# B&R Automation Studio project Genmot_Markalama_ (part 5)

#### GRYAxisControl.c - Implementation code
```c
/*******************************************************************
 * COPYRIGHT -- Bernecker + Rainer
 ********************************************************************
 * PROGRAM: Basic
 * File: Basic.c
 * Author: Bernecker + Rainer
 * Created: December 01, 2009
 ********************************************************************
 * Implementation of Program Basic
 ********************************************************************/

#ifdef _DEFAULT_INCLUDES
#include <AsDefault.h>
#endif
#include <string.h>

/* defines of the state-constants */
#define STATE_WAIT              0
#define STATE_POWER_ON          1
#define STATE_HOME              2

#define STATE_READY             10
#define STATE_HALT              11
#define STATE_STOP              12
#define STATE_JOG_POSITIVE      13
#define STATE_JOG_NEGATIVE      14
#define STATE_MOVE_ABSOLUTE     15
#define STATE_MOVE_ADDITIVE     16
#define STATE_MOVE_VELOCITY     17

#define STATE_ERROR_AXIS        100
#define STATE_ERROR             101
#define STATE_ERROR_RESET       102
#define STATE_READ              103

_LOCAL REAL   data;

_INIT void GRYAxis_init(void)
{

	/* get axis object */
	Axis1Obj = (UDINT)&GRY_Axis;

	AxisStep = STATE_WAIT;  /* start step */

	GRYAxis.Parameter.Velocity              = 10000;  /*velocity for movement*/
	GRYAxis.Parameter.Acceleration          = 40000;  /*acceleration for movement*/
	GRYAxis.Parameter.Deceleration          = 40000;  /*deceleration for movement*/
	GRYAxis.Parameter.JogVelocity           = 10000;   /*velocity for jogging */

}

_CYCLIC void GRYAxis_cyclic(void)
{
	if(GRYAxis.Command.Power)
	{
		GRYAxis.Speed.VelocityOverride			= 1.0;
	}

/***************************************************************
        Control Sequence
***************************************************************/

/* status information is read before the step sequencer to attain a shorter reaction time */
/************************ MC_READSTATUS *************************/
	MC_ReadStatus_0.Enable = !MC_ReadStatus_0.Error;
	MC_ReadStatus_0.Axis = Axis1Obj;
	MC_ReadStatus(&MC_ReadStatus_0);
	GRYAxis.AxisState.Disabled             = MC_ReadStatus_0.Disabled;
	GRYAxis.AxisState.StandStill           = MC_ReadStatus_0.StandStill;
	GRYAxis.AxisState.Stopping             = MC_ReadStatus_0.Stopping;
	GRYAxis.AxisState.Homing               = MC_ReadStatus_0.Homing;
	GRYAxis.AxisState.DiscreteMotion       = MC_ReadStatus_0.DiscreteMotion;
	GRYAxis.AxisState.ContinuousMotion     = MC_ReadStatus_0.ContinuousMotion;
	GRYAxis.AxisState.SynchronizedMotion   = MC_ReadStatus_0.SynchronizedMotion;
	GRYAxis.AxisState.ErrorStop            = MC_ReadStatus_0.Errorstop;

	/********************MC_BR_READDRIVESTATUS***********************/
	MC_BR_ReadDriveStatus_0.Enable = !MC_BR_ReadDriveStatus_0.Error;
	MC_BR_ReadDriveStatus_0.Axis = Axis1Obj;
	MC_BR_ReadDriveStatus_0.AdrDriveStatus = (UDINT)&(GRYAxis.Status.DriveStatus);
	MC_BR_ReadDriveStatus(&MC_BR_ReadDriveStatus_0);

	/******************** MC_READACTUALPOSITION *********************/
	MC_ReadActualPosition_0.Enable = (!MC_ReadActualPosition_0.Error);
	MC_ReadActualPosition_0.Axis = Axis1Obj;
	MC_ReadActualPosition(&MC_ReadActualPosition_0);
	if(MC_ReadActualPosition_0.Valid == 1)
	{
		GRYAxis.Status.ActPosition = MC_ReadActualPosition_0.Position;
	}

	/******************** MC_READACTUALVELOCITY *********************/
	MC_ReadActualVelocity_0.Enable = (!MC_ReadActualVelocity_0.Error);
	MC_ReadActualVelocity_0.Axis = Axis1Obj;
	MC_ReadActualVelocity(&MC_ReadActualVelocity_0);
	if(MC_ReadActualVelocity_0.Valid == 1)
	{
		GRYAxis.Status.ActVelocity = MC_ReadActualVelocity_0.Velocity;
	}

	/*********************** MC SET OVERRIDE *********************/
	MC_SetOverride_0.Enable = (!MC_SetOverride_0.Error);
	MC_SetOverride_0.AccFactor = GRYAxis.Speed.AccelerationOverride = 1.0;
	if ((GRYAxis.Speed.VelocityOverride < 2.01) && (GRYAxis.Speed.VelocityOverride > 0.0000001))
	{
		MC_SetOverride_0.VelFactor = GRYAxis.Speed.VelocityOverride;
	}
	MC_SetOverride_0.Axis=Axis1Obj;
	MC_SetOverride(&MC_SetOverride_0);

	/************************ MC_READAXISERROR **********************/
	MC_ReadAxisError_0.Enable = !MC_ReadAxisError_0.Error;
	MC_ReadAxisError_0.Axis = Axis1Obj;
	MC_ReadAxisError_0.DataAddress = (UDINT)&(GRYAxis.Status.ErrorText);
	MC_ReadAxisError_0.DataLength = sizeof(GRYAxis.Status.ErrorText);
	strcpy((void*)&MC_ReadAxisError_0.DataObjectName,"acp10etxen");
	MC_ReadAxisError(&MC_ReadAxisError_0);

	/* central monitoring of stop command attains a shorter reaction time in case of emergency stop */
	/******************CHECK for STOP COMMAND************************/
	if (GRYAxis.Command.Stop == 1)
	{
		if ((AxisStep >= STATE_READY) && (AxisStep < STATE_ERROR))
		{
			/* reset all FB execute inputs we use */
			MC_Home_0.Execute = 0;
			MC_Stop_0.Execute = 0;
			MC_MoveAbsolute_0.Execute = 0;
			MC_MoveAdditive_0.Execute = 0;
			MC_MoveVelocity_0.Execute = 0;
			MC_ReadAxisError_0.Acknowledge = 0;
			MC_Reset_0.Execute = 0;

			/* reset user commands */
			GRYAxis.Command.Stop = 0;
			GRYAxis.Command.Home = 0;
			GRYAxis.Command.MoveJogPos = 0;
			GRYAxis.Command.MoveJogNeg = 0;
			GRYAxis.Command.MoveVelocity = 0;
			GRYAxis.Command.MoveAbsolute = 0;
			GRYAxis.Command.MoveAdditive = 0;
			AxisStep = STATE_STOP;
		}
	}

	/**************** CHECK FOR GENERAL AXIS ERROR ******************/
	if ((MC_ReadAxisError_0.AxisErrorID != 0) && (MC_ReadAxisError_0.Valid == 1))
	{
		AxisStep = STATE_ERROR_AXIS;
	}
		/***************** CHECK IF POWER SHOULD BE OFF *******************/
	else if ((GRYAxis.Command.Power == 0) && (MC_ReadAxisError_0.Valid == 1))
	{
		if ((MC_ReadStatus_0.Errorstop == 1) && (MC_ReadStatus_0.Valid == 1))
		{
			AxisStep = STATE_ERROR_RESET;
		}
		else
		{
			AxisStep = STATE_WAIT;
		}
	}

	switch(AxisStep)
	{
		/******************** WAIT *************************/
		case STATE_WAIT:  /* STATE: Wait */
			if (GRYAxis.Command.Power == 1)
			{
				AxisStep = STATE_POWER_ON;
			}
			else
			{
				MC_Power_0.Enable = 0;

			}

			/* reset all FB execute inputs we use */
			MC_Home_0.Execute = 0;
			MC_Stop_0.Execute = 0;
			MC_MoveAbsolute_0.Execute = 0;
			MC_MoveAdditive_0.Execute = 0;
			MC_MoveVelocity_0.Execute = 0;
			MC_ReadAxisError_0.Acknowledge = 0;
			MC_Reset_0.Execute = 0;

			/* reset user commands */
			GRYAxis.Command.Stop = 0;
			GRYAxis.Command.Home = 0;
			GRYAxis.Command.MoveJogPos = 0;
			GRYAxis.Command.MoveJogNeg = 0;
			GRYAxis.Command.MoveVelocity = 0;
			GRYAxis.Command.MoveAbsolute = 0;
			GRYAxis.Command.MoveAdditive = 0;

			GRYAxis.Status.ErrorID = 0;
			break;

		/******************** POWER ON **********************/
		case STATE_POWER_ON:  /* STATE: Power on */
			MC_Power_0.Enable = 1;
			if (MC_Power_0.Status == 1)
			{
			if (!GRXHomeOk)
			{
			GRYAxis.Command.Home = 1;
			}
			AxisStep = STATE_READY;
			}
			/* if a power error occured go to error state */
			if (MC_Power_0.Error == 1)
			{
				GRYAxis.Status.ErrorID = MC_Power_0.ErrorID;
				AxisStep = STATE_ERROR;
			}
			break;

		/******************** READY **********************/
		case STATE_READY:  /* STATE: Waiting for commands */
			if (GRYAxis.Command.Home == 1)
			{
				GRYAxis.Command.Home = 0;
				AxisStep = STATE_HOME;
			}
			else if (GRYAxis.Command.Stop == 1)
			{
				AxisStep = STATE_STOP;
			}
			else if (GRYAxis.Command.MoveJogPos == 1)
			{
				AxisStep = STATE_JOG_POSITIVE;
			}
			else if (GRYAxis.Command.MoveJogNeg == 1)
			{
				AxisStep = STATE_JOG_NEGATIVE;
			}
			else if (GRYAxis.Command.MoveAbsolute == 1)
			{
				GRYAxis.Command.MoveAbsolute = 0;
				AxisStep = STATE_MOVE_ABSOLUTE;
			}
			else if (GRYAxis.Command.MoveAdditive == 1)
			{
				GRYAxis.Command.MoveAdditive = 0;
				AxisStep = STATE_MOVE_ADDITIVE;
			}
			else if (GRYAxis.Command.MoveVelocity == 1)
			{
				GRYAxis.Command.MoveVelocity = 0;
				AxisStep = STATE_MOVE_VELOCITY;
			}
			else if (GRYAxis.Command.Halt == 1)
			{
				GRYAxis.Command.Halt = 0;
				AxisStep = STATE_HALT;
			}
			break;

		/******************** HOME **********************/
		case STATE_HOME:  /* STATE: start homing process */
			MC_Home_0.Position = GRYAxis.Parameter.HomePosition;
			MC_Home_0.HomingMode = GRYAxis.Parameter.HomeMode;
			MC_Home_0.Execute = 1;
			if (MC_Home_0.Done == 1)
			{

				MC_Home_0.Execute = 0;
				AxisStep = STATE_READ;
			}
			/* if a homing error occured go to error state */
			if (MC_Home_0.Error == 1)
			{
				MC_Home_0.Execute = 0;
				GRYAxis.Status.ErrorID = MC_Home_0.ErrorID;
				AxisStep = STATE_ERROR;
			}
			break;

		/************************HALT MOVEMENT**************************/
		case STATE_HALT:  /* STATE: Stop the active movement */
			MC_Halt_0.Deceleration = GRYAxis.Parameter.Deceleration;
			MC_Halt_0.Execute = 1;
			if (MC_Halt_0.Done == 1)
			{
				MC_Halt_0.Execute = 0;
				AxisStep = STATE_READY;
			}
			/*check if error occured */
			if (MC_Halt_0.Error == 1)
			{
				MC_Halt_0.Execute = 0;
				GRYAxis.Status.ErrorID = MC_Halt_0.ErrorID;
				AxisStep = STATE_ERROR;
			}
			break;

		/*********************** STOP MOVEMENT *************************/
		case STATE_STOP: /* STATE: Stop movement as long as command is set */
			MC_Stop_0.Deceleration = GRYAxis.Parameter.Deceleration;
			MC_Stop_0.Execute = 1;
			/* if axis is stopped go to ready state */
			if ((MC_Stop_0.Done == 1) && (GRYAxis.Command.Stop == 0))
			{
				MC_Stop_0.Execute = 0;
				AxisStep = STATE_READY;
			}
			/* check if error occured */
			if (MC_Stop_0.Error == 1)
			{
				GRYAxis.Status.ErrorID = MC_Stop_0.ErrorID;
				MC_Stop_0.Execute = 0;
				AxisStep = STATE_ERROR;
			}
			break;

		/******************** START JOG MOVEMENT POSITVE **********************/
		case STATE_JOG_POSITIVE:  /* STATE: Start jog movement in positive direction */
			MC_MoveVelocity_0.Velocity      = GRYAxis.Parameter.JogVelocity;
			MC_MoveVelocity_0.Acceleration  = GRYAxis.Parameter.Acceleration;
			MC_MoveVelocity_0.Deceleration  = GRYAxis.Parameter.Deceleration;
			MC_MoveVelocity_0.Direction     = mcPOSITIVE_DIR;
			MC_MoveVelocity_0.Execute = 1;
			/* check if jog movement should be stopped */
			if (GRYAxis.Command.MoveJogPos == 0)
			{
				MC_MoveVelocity_0.Execute = 0;
				AxisStep = STATE_HALT;
			}
			/* check if error occured */
			if (MC_MoveVelocity_0.Error == 1)
			{
				GRYAxis.Status.ErrorID = MC_MoveVelocity_0.ErrorID;
				MC_MoveVelocity_0.Execute = 0;
				AxisStep = STATE_ERROR;
			}
			break;

		/******************** START JOG MOVEMENT NEGATIVE **********************/
		case STATE_JOG_NEGATIVE:  /* STATE: Start jog movement in negative direction */
			MC_MoveVelocity_0.Velocity      = GRYAxis.Parameter.JogVelocity;
			MC_MoveVelocity_0.Acceleration  = GRYAxis.Parameter.Acceleration;
			MC_MoveVelocity_0.Deceleration  = GRYAxis.Parameter.Deceleration;
			MC_MoveVelocity_0.Direction     = mcNEGATIVE_DIR;
			MC_MoveVelocity_0.Execute = 1;
			/* check if jog movement should be stopped */
			if (GRYAxis.Command.MoveJogNeg == 0)
			{
				MC_MoveVelocity_0.Execute = 0;
				AxisStep = STATE_HALT;
			}
			/* check if error occured */
			if (MC_MoveVelocity_0.Error == 1)
			{
				GRYAxis.Status.ErrorID = MC_MoveVelocity_0.ErrorID;
				MC_MoveVelocity_0.Execute = 0;
				AxisStep = STATE_ERROR;
			}
			break;

		/******************** START ABSOLUTE MOVEMENT **********************/
		case STATE_MOVE_ABSOLUTE:  /* STATE: Start absolute movement */
			MC_MoveAbsolute_0.Position      = GRYAxis.Parameter.Position;
			MC_MoveAbsolute_0.Velocity      = GRYAxis.Parameter.Velocity;
			MC_MoveAbsolute_0.Acceleration  = GRYAxis.Parameter.Acceleration;
			MC_MoveAbsolute_0.Deceleration  = GRYAxis.Parameter.Deceleration;
			MC_MoveAbsolute_0.Direction     = GRYAxis.Parameter.Direction;
			MC_MoveAbsolute_0.Execute = 1;
			/* check if commanded position is reached */
			if (GRYAxis.Command.Halt == 1)
			{
				GRYAxis.Command.Halt = 0;
				MC_MoveAbsolute_0.Execute = 0;
				AxisStep = STATE_HALT;
			}
			else if (MC_MoveAbsolute_0.Done == 1)
			{
				MC_MoveAbsolute_0.Execute = 0;
				AxisStep = STATE_READY;
			}
			/* check if error occured */
			if (MC_MoveAbsolute_0.Error == 1)
			{
				GRYAxis.Status.ErrorID = MC_MoveAbsolute_0.ErrorID;
				MC_MoveAbsolute_0.Execute = 0;
				AxisStep = STATE_ERROR;
			}
			break;

		/******************** START ADDITIVE MOVEMENT **********************/
		case STATE_MOVE_ADDITIVE:  /* STATE: Start additive movement */
			MC_MoveAdditive_0.Distance      = GRYAxis.Parameter.Distance;
			MC_MoveAdditive_0.Velocity      = GRYAxis.Parameter.Velocity;
			MC_MoveAdditive_0.Acceleration  = GRYAxis.Parameter.Acceleration;
			MC_MoveAdditive_0.Deceleration  = GRYAxis.Parameter.Deceleration;
			MC_MoveAdditive_0.Execute = 1;
			/* check if commanded distance is reached */
			if (GRYAxis.Command.Halt == 1)
			{
				GRYAxis.Command.Halt = 0;
				MC_MoveAdditive_0.Execute = 0;
				AxisStep = STATE_HALT;
			}
			else if (MC_MoveAdditive_0.Done == 1)
			{
				MC_MoveAdditive_0.Execute = 0;
				AxisStep = STATE_READY;
			}
			/* check if error occured */
			if (MC_MoveAdditive_0.Error == 1)
			{
				GRYAxis.Status.ErrorID = MC_MoveAdditive_0.ErrorID;
				MC_MoveAdditive_0.Execute = 0;
				AxisStep = STATE_ERROR;
			}
			break;

		/******************** START VELOCITY MOVEMENT **********************/
		case STATE_MOVE_VELOCITY:  /* STATE: Start velocity movement */
			MC_MoveVelocity_0.Velocity      = GRYAxis.Parameter.Velocity;
			MC_MoveVelocity_0.Acceleration  = GRYAxis.Parameter.Acceleration;
			MC_MoveVelocity_0.Deceleration  = GRYAxis.Parameter.Deceleration;
			MC_MoveVelocity_0.Direction     = GRYAxis.Parameter.Direction;
			MC_MoveVelocity_0.Execute = 1;
			/* check if commanded velocity is reached */
			if (GRYAxis.Command.Halt == 1)
			{
				GRYAxis.Command.Halt = 0;
				MC_MoveVelocity_0.Execute = 0;
				AxisStep = STATE_HALT;
			}
			else if (MC_MoveVelocity_0.InVelocity == 1)
			{
				MC_MoveVelocity_0.Execute = 0;
				AxisStep = STATE_READY;
			}
			/* check if error occured */
			if (MC_MoveVelocity_0.Error == 1)
			{
				GRYAxis.Status.ErrorID = MC_MoveVelocity_0.ErrorID;
				MC_MoveVelocity_0.Execute = 0;
				AxisStep = STATE_ERROR;
			}
			break;

		/******************** FB-ERROR OCCURED *************************/
		case STATE_ERROR:  /* STATE: Error */
			/* check if FB indicates an axis error */
			if (MC_ReadAxisError_0.AxisErrorCount != 0)
			{
				AxisStep = STATE_ERROR_AXIS;
			}
			else
			{
				if (GRYAxis.Command.ErrorAcknowledge == 1)
				{
					GRYAxis.Command.ErrorAcknowledge = 0;
					GRYAxis.Status.ErrorID = 0;
					/* reset axis if it is in axis state ErrorStop */
					if ((MC_ReadStatus_0.Errorstop == 1) && (MC_ReadStatus_0.Valid == 1))
					{
						AxisStep = STATE_ERROR_RESET;
					}
					else
					{
						AxisStep = STATE_WAIT;
					}
				}
			}
			break;

		/******************** AXIS-ERROR OCCURED *************************/
		case STATE_ERROR_AXIS:  /* STATE: Axis Error */
			if (MC_ReadAxisError_0.Valid == 1)
			{
				if (MC_ReadAxisError_0.AxisErrorID != 0)
				{
					GRYAxis.Status.ErrorID = MC_ReadAxisError_0.AxisErrorID;
				}
				MC_ReadAxisError_0.Acknowledge = 0;
				if (GRYAxis.Command.ErrorAcknowledge == 1)
				{
					GRYAxis.Command.ErrorAcknowledge = 0;
					/* acknowledge axis error */
					if (MC_ReadAxisError_0.AxisErrorID != 0)
					{
						MC_ReadAxisError_0.Acknowledge = 1;
					}
				}
				if (MC_ReadAxisError_0.AxisErrorCount == 0)
				{
					GRYAxis.Status.ErrorID = 0;
					/* reset axis if it is in axis state ErrorStop */
					if ((MC_ReadStatus_0.Errorstop == 1) && (MC_ReadStatus_0.Valid == 1))
					{
						AxisStep = STATE_ERROR_RESET;
					}
					else
					{
						AxisStep = STATE_WAIT;
					}
				}
			}
			break;

		/******************** RESET DONE *************************/
		case STATE_ERROR_RESET:  /* STATE: Wait for reset done */
			MC_Reset_0.Execute = 1;
			/* reset MC_Power.Enable if this FB is in Error*/
			if(MC_Power_0.Error == 1)
			{
				MC_Power_0.Enable = 0;
			}
			if(MC_Reset_0.Done == 1)
			{
				MC_Reset_0.Execute = 0;
				AxisStep = STATE_WAIT;
			}
			else if (MC_Reset_0.Error == 1)
			{
				MC_Reset_0.Execute = 0;
				AxisStep = STATE_ERROR;
			}
			break;

		/******************** SEQUENCE END *************************/

		/**********************STATE_READ************************/
		case STATE_READ:
			MC_BR_CyclicRead_0.Enable=1;
			MC_BR_CyclicRead_0.ParID = 277;
			MC_BR_CyclicRead_0.DataAddress = (UDINT)&data;
			MC_BR_CyclicRead_0.DataType =ncPAR_TYP_REAL;

			if (MC_BR_CyclicRead_0.Valid)
			{
				AxisStep = STATE_READY;
			}
			else if (MC_BR_CyclicRead_0.Error)
			{

				GRYAxis.Status.ErrorID = MC_BR_CyclicRead_0.ErrorID;
				/*Reset Enable before going to STATE_ERROR*/
				MC_BR_CyclicRead_0.Enable=0;
				AxisStep = STATE_ERROR;
			}
			break;  /*end read*/

	}

/***************************************************************
        Function Block Calls
***************************************************************/

/************************** MC_POWER ****************************/
	MC_Power_0.Axis = Axis1Obj;  /* pointer to axis */
	MC_Power(&MC_Power_0);

	/************************** MC_HOME *****************************/
	MC_Home_0.Axis = Axis1Obj;
	MC_Home(&MC_Home_0);

	/********************** MC_MOVEABSOLUTE *************************/
	MC_MoveAbsolute_0.Axis = Axis1Obj;
	MC_MoveAbsolute(&MC_MoveAbsolute_0);

	/********************** MC_MOVEADDITIVE *************************/
	MC_MoveAdditive_0.Axis = Axis1Obj;
	MC_MoveAdditive(&MC_MoveAdditive_0);

	/********************** MC_MOVEVELOCITY *************************/
	MC_MoveVelocity_0.Axis = Axis1Obj;
	MC_MoveVelocity(&MC_MoveVelocity_0);

	/************************** MC_STOP *****************************/
	MC_Stop_0.Axis = Axis1Obj;
	MC_Stop(&MC_Stop_0);

	/**************************MC_HALT*******************************/
	MC_Halt_0.Axis = Axis1Obj;
	MC_Halt(&MC_Halt_0);

	/************************** MC_RESET ****************************/
	MC_Reset_0.Axis = Axis1Obj;
	MC_Reset(&MC_Reset_0);

	MC_BR_CyclicRead_0.Axis = Axis1Obj;
	MC_BR_CyclicRead(&MC_BR_CyclicRead_0);

}
```

#### GRYAxisControl.var - Local variables
```iecst
(********************************************************************
 * COPYRIGHT --
 ********************************************************************
 * Program: Reg2Ax
 * File: Reg2Ax.var
 * Author: Coder
 * Created: June 20, 2013
 ********************************************************************
 * Local variables of program Reg2Ax
 ********************************************************************)
VAR
	Axis1Obj : UDINT; (*axis reference*)
	Axis2Obj : UDINT; (*axis reference*)
	AxisStep : USINT; (*current step in the step sequence*)
	AutData : MC_AUTDATA_TYP := (0); (*configuration of the automat*)
	MC_Power_0 : MC_Power; (*Function Block*)
	MC_Home_0 : MC_Home; (*Function Block*)
	MC_Stop_0 : MC_Stop; (*Function Block*)
	MC_MoveVelocity_0 : MC_MoveVelocity; (*Function Block*)
	MC_MoveAbsolute_0 : MC_MoveAbsolute; (*Function Block*)
	MC_MoveAdditive_0 : MC_MoveAdditive; (*Function Block*)
	MC_BR_InitAutData_0 : MC_BR_InitAutData; (*Function Block*)
	MC_BR_AutControl_0 : MC_BR_AutControl; (*Function Block*)
	MC_ReadAxisError_0 : MC_ReadAxisError; (*Function Block*)
	MC_Reset_0 : MC_Reset; (*Function Block*)
	MC_ReadStatus_0 : MC_ReadStatus; (*Function Block*)
	MC_ReadActualPosition_0 : MC_ReadActualPosition; (*Function Block*)
	MC_ReadActualVelocity_0 : MC_ReadActualVelocity; (*Function Block*)
	MC_BR_ReadDriveStatus_0 : MC_BR_ReadDriveStatus; (*Function Block*)
	MC_Halt_0 : MC_Halt; (*Function Block*)
	MC_BR_DownloadCamProfileObj_0 : MC_BR_DownloadCamProfileObj;
	SlaveFactor : REAL;
	MC_BR_Phasing_0 : MC_BR_Phasing;
	ShiftFactor : REAL;
	MC_GearInPos_0 : MC_GearInPos;
	MC_GearOut_0 : MC_GearOut;
	MC_SetOverride_0 : MC_SetOverride;
	MC_BR_CyclicRead_0 : MC_BR_CyclicRead;
END_VAR
(********************************************************************
 * COPYRIGHT --
 ********************************************************************
 * Program: GRYAxisControl
 * File: GRYAxisControl.var
 * Author: Administrator
 * Created: September 22, 2017
 ********************************************************************
 * Local variables of program GRYAxisControl
 ********************************************************************)
```

#### edge.h
```c
/*
	edge.h

	Macros for Edgedetection. This macros uses a special feature of the GNU compiler:
	"Statements and Declarations in Expressions" see more details in GNU-Documentation
	So they may not work with other compilers.

	EDGEPOS  return 1 at positive transition of signal, in all other cases 0 is returned
	EDGENEG  return 1 at negative transition of signal, in all other cases 0 is returned
	EDGEPOS  return 1 at positive and negative transition of signal, in all other cases 0 is returned
*/

#ifndef __EDGE_H__
#define __EDGE_H__

#define EDGEPOS(variable) ({static plcbit __oldval=0; plcbit result; \
                            if (variable && !__oldval)               \
                              result=1;                              \
                            else                                     \
                              result=0;                              \
                              __oldval=variable;                     \
                              result;                                \
                           })

#define EDGENEG(variable) ({static plcbit __oldval=0; plcbit result; \
                            if (!variable && __oldval)               \
                              result=1;                              \
                            else                                     \
                              result=0;                              \
                              __oldval=variable;                     \
                              result;                                \
                           })

#define EDGE(variable)    ({static plcbit __oldval=0; plcbit result; \
                            if (variable != __oldval)                \
                              result=1;                              \
                            else                                     \
                              result=0;                              \
                              __oldval=variable;                     \
                              result;                                \
                           })

#endif /*__EDGE_H__*/
```

### Program Logical/GRZAxisControl (ANSIC)

#### GRZAx.c - Implementation code
```c
/*******************************************************************
 * COPYRIGHT -- Bernecker + Rainer
 ********************************************************************
 * PROGRAM: Basic
 * File: Basic.c
 * Author: Bernecker + Rainer
 * Created: December 01, 2009
 ********************************************************************
 * Implementation of Program Basic
 ********************************************************************/

#ifdef _DEFAULT_INCLUDES
#include <AsDefault.h>
#endif
#include <string.h>

/* defines of the state-constants */
#define STATE_WAIT              0
#define STATE_POWER_ON          1
#define STATE_HOME              2

#define STATE_READY             10
#define STATE_HALT              11
#define STATE_STOP              12
#define STATE_JOG_POSITIVE      13
#define STATE_JOG_NEGATIVE      14
#define STATE_MOVE_ABSOLUTE     15
#define STATE_MOVE_ADDITIVE     16
#define STATE_MOVE_VELOCITY     17

#define STATE_ERROR_AXIS        100
#define STATE_ERROR             101
#define STATE_ERROR_RESET       102
#define STATE_READ              103

_LOCAL REAL   data;

_INIT void GRZAxis_init(void)
{

	/* get axis object */
	Axis1Obj = (UDINT)&GRZ_Axis;

	AxisStep = STATE_WAIT;  /* start step */

	GRZAxis.Parameter.Velocity              = 40000;  /*velocity for movement*/
	GRZAxis.Parameter.Acceleration          = 120000;  /*acceleration for movement*/
	GRZAxis.Parameter.Deceleration          = 120000;  /*deceleration for movement*/
	GRZAxis.Parameter.JogVelocity           = 40000;   /*velocity for jogging */

}

_CYCLIC void GRZAxis_cyclic(void)
{
	if(GRZAxis.Command.Power)
	{
		GRZAxis.Speed.VelocityOverride			= 1.0;
	}

/***************************************************************
        Control Sequence
***************************************************************/

/* status information is read before the step sequencer to attain a shorter reaction time */
/************************ MC_READSTATUS *************************/
	MC_ReadStatus_0.Enable = !MC_ReadStatus_0.Error;
	MC_ReadStatus_0.Axis = Axis1Obj;
	MC_ReadStatus(&MC_ReadStatus_0);
	GRZAxis.AxisState.Disabled             = MC_ReadStatus_0.Disabled;
	GRZAxis.AxisState.StandStill           = MC_ReadStatus_0.StandStill;
	GRZAxis.AxisState.Stopping             = MC_ReadStatus_0.Stopping;
	GRZAxis.AxisState.Homing               = MC_ReadStatus_0.Homing;
	GRZAxis.AxisState.DiscreteMotion       = MC_ReadStatus_0.DiscreteMotion;
	GRZAxis.AxisState.ContinuousMotion     = MC_ReadStatus_0.ContinuousMotion;
	GRZAxis.AxisState.SynchronizedMotion   = MC_ReadStatus_0.SynchronizedMotion;
	GRZAxis.AxisState.ErrorStop            = MC_ReadStatus_0.Errorstop;

	/********************MC_BR_READDRIVESTATUS***********************/
	MC_BR_ReadDriveStatus_0.Enable = !MC_BR_ReadDriveStatus_0.Error;
	MC_BR_ReadDriveStatus_0.Axis = Axis1Obj;
	MC_BR_ReadDriveStatus_0.AdrDriveStatus = (UDINT)&(GRZAxis.Status.DriveStatus);
	MC_BR_ReadDriveStatus(&MC_BR_ReadDriveStatus_0);

	/******************** MC_READACTUALPOSITION *********************/
	MC_ReadActualPosition_0.Enable = (!MC_ReadActualPosition_0.Error);
	MC_ReadActualPosition_0.Axis = Axis1Obj;
	MC_ReadActualPosition(&MC_ReadActualPosition_0);
	if(MC_ReadActualPosition_0.Valid == 1)
	{
		GRZAxis.Status.ActPosition = MC_ReadActualPosition_0.Position;
	}

	/******************** MC_READACTUALVELOCITY *********************/
	MC_ReadActualVelocity_0.Enable = (!MC_ReadActualVelocity_0.Error);
	MC_ReadActualVelocity_0.Axis = Axis1Obj;
	MC_ReadActualVelocity(&MC_ReadActualVelocity_0);
	if(MC_ReadActualVelocity_0.Valid == 1)
	{
		GRZAxis.Status.ActVelocity = MC_ReadActualVelocity_0.Velocity;
	}

	/*********************** MC SET OVERRIDE *********************/
	MC_SetOverride_0.Enable = (!MC_SetOverride_0.Error);
	MC_SetOverride_0.AccFactor = GRZAxis.Speed.AccelerationOverride = 1.0;
	if ((GRZAxis.Speed.VelocityOverride < 2.01) && (GRZAxis.Speed.VelocityOverride > 0.0000001))
	{
		MC_SetOverride_0.VelFactor = GRZAxis.Speed.VelocityOverride;
	}
	MC_SetOverride_0.Axis=Axis1Obj;
	MC_SetOverride(&MC_SetOverride_0);

	/************************ MC_READAXISERROR **********************/
	MC_ReadAxisError_0.Enable = !MC_ReadAxisError_0.Error;
	MC_ReadAxisError_0.Axis = Axis1Obj;
	MC_ReadAxisError_0.DataAddress = (UDINT)&(GRZAxis.Status.ErrorText);
	MC_ReadAxisError_0.DataLength = sizeof(GRZAxis.Status.ErrorText);
	strcpy((void*)&MC_ReadAxisError_0.DataObjectName,"acp10etxen");
	MC_ReadAxisError(&MC_ReadAxisError_0);

	/* central monitoring of stop command attains a shorter reaction time in case of emergency stop */
	/******************CHECK for STOP COMMAND************************/
	if (GRZAxis.Command.Stop == 1)
	{
		if ((AxisStep >= STATE_READY) && (AxisStep < STATE_ERROR))
		{
			/* reset all FB execute inputs we use */
			MC_Home_0.Execute = 0;
			MC_Stop_0.Execute = 0;
			MC_MoveAbsolute_0.Execute = 0;
			MC_MoveAdditive_0.Execute = 0;
			MC_MoveVelocity_0.Execute = 0;
			MC_ReadAxisError_0.Acknowledge = 0;
			MC_Reset_0.Execute = 0;

			/* reset user commands */
			GRZAxis.Command.Stop = 0;
			GRZAxis.Command.Home = 0;
			GRZAxis.Command.MoveJogPos = 0;
			GRZAxis.Command.MoveJogNeg = 0;
			GRZAxis.Command.MoveVelocity = 0;
			GRZAxis.Command.MoveAbsolute = 0;
			GRZAxis.Command.MoveAdditive = 0;
			AxisStep = STATE_STOP;
		}
	}

	/**************** CHECK FOR GENERAL AXIS ERROR ******************/
	if ((MC_ReadAxisError_0.AxisErrorID != 0) && (MC_ReadAxisError_0.Valid == 1))
	{
		AxisStep = STATE_ERROR_AXIS;
	}
		/***************** CHECK IF POWER SHOULD BE OFF *******************/
	else if ((GRZAxis.Command.Power == 0) && (MC_ReadAxisError_0.Valid == 1))
	{
		if ((MC_ReadStatus_0.Errorstop == 1) && (MC_ReadStatus_0.Valid == 1))
		{
			AxisStep = STATE_ERROR_RESET;
		}
		else
		{
			AxisStep = STATE_WAIT;
		}
	}

	switch(AxisStep)
	{
		/******************** WAIT *************************/
		case STATE_WAIT:  /* STATE: Wait */
			if (GRZAxis.Command.Power == 1)
			{
				AxisStep = STATE_POWER_ON;
			}
			else
			{
				MC_Power_0.Enable = 0;

			}

			/* reset all FB execute inputs we use */
			MC_Home_0.Execute = 0;
			MC_Stop_0.Execute = 0;
			MC_MoveAbsolute_0.Execute = 0;
			MC_MoveAdditive_0.Execute = 0;
			MC_MoveVelocity_0.Execute = 0;
			MC_ReadAxisError_0.Acknowledge = 0;
			MC_Reset_0.Execute = 0;

			/* reset user commands */
			GRZAxis.Command.Stop = 0;
			GRZAxis.Command.Home = 0;
			GRZAxis.Command.MoveJogPos = 0;
			GRZAxis.Command.MoveJogNeg = 0;
			GRZAxis.Command.MoveVelocity = 0;
			GRZAxis.Command.MoveAbsolute = 0;
			GRZAxis.Command.MoveAdditive = 0;

			GRZAxis.Status.ErrorID = 0;
			break;

		/******************** POWER ON **********************/
		case STATE_POWER_ON:  /* STATE: Power on */
			MC_Power_0.Enable = 1;
			if (MC_Power_0.Status == 1)
			{
				if (!GRZHomeOk)
				{
					GRZAxis.Command.Home = 1;
				}
			    AxisStep = STATE_READY;
			}
			/* if a power error occured go to error state */
			if (MC_Power_0.Error == 1)
			{
				GRZAxis.Status.ErrorID = MC_Power_0.ErrorID;
				AxisStep = STATE_ERROR;
			}
			break;

		/******************** READY **********************/
		case STATE_READY:  /* STATE: Waiting for commands */
			if (GRZAxis.Command.Home == 1)
			{
				GRZAxis.Command.Home = 0;
				AxisStep = STATE_HOME;
			}
			else if (GRZAxis.Command.Stop == 1)
			{
				AxisStep = STATE_STOP;
			}
			else if (GRZAxis.Command.MoveJogPos == 1)
			{
				AxisStep = STATE_JOG_POSITIVE;
			}
			else if (GRZAxis.Command.MoveJogNeg == 1)
			{
				AxisStep = STATE_JOG_NEGATIVE;
			}
			else if (GRZAxis.Command.MoveAbsolute == 1)
			{
				GRZAxis.Command.MoveAbsolute = 0;
				AxisStep = STATE_MOVE_ABSOLUTE;
			}
			else if (GRZAxis.Command.MoveAdditive == 1)
			{
				GRZAxis.Command.MoveAdditive = 0;
				AxisStep = STATE_MOVE_ADDITIVE;
			}
			else if (GRZAxis.Command.MoveVelocity == 1)
			{
				GRZAxis.Command.MoveVelocity = 0;
				AxisStep = STATE_MOVE_VELOCITY;
			}
			else if (GRZAxis.Command.Halt == 1)
			{
				GRZAxis.Command.Halt = 0;
				AxisStep = STATE_HALT;
			}
			break;

		/******************** HOME **********************/
		case STATE_HOME:  /* STATE: start homing process */
			MC_Home_0.Position = GRZAxis.Parameter.HomePosition;
			MC_Home_0.HomingMode = GRZAxis.Parameter.HomeMode;
			MC_Home_0.Execute = 1;
			if (MC_Home_0.Done == 1)
			{

				MC_Home_0.Execute = 0;
				AxisStep = STATE_READ;
			}
			/* if a homing error occured go to error state */
			if (MC_Home_0.Error == 1)
			{
				MC_Home_0.Execute = 0;
				GRZAxis.Status.ErrorID = MC_Home_0.ErrorID;
				AxisStep = STATE_ERROR;
			}
			break;

		/************************HALT MOVEMENT**************************/
		case STATE_HALT:  /* STATE: Stop the active movement */
			MC_Halt_0.Deceleration = GRZAxis.Parameter.Deceleration;
			MC_Halt_0.Execute = 1;
			if (MC_Halt_0.Done == 1)
			{
				MC_Halt_0.Execute = 0;
				AxisStep = STATE_READY;
			}
			/*check if error occured */
			if (MC_Halt_0.Error == 1)
			{
				MC_Halt_0.Execute = 0;
				GRZAxis.Status.ErrorID = MC_Halt_0.ErrorID;
				AxisStep = STATE_ERROR;
			}
			break;

		/*********************** STOP MOVEMENT *************************/
		case STATE_STOP: /* STATE: Stop movement as long as command is set */
			MC_Stop_0.Deceleration = GRZAxis.Parameter.Deceleration;
			MC_Stop_0.Execute = 1;
			/* if axis is stopped go to ready state */
			if ((MC_Stop_0.Done == 1) && (GRZAxis.Command.Stop == 0))
			{
				MC_Stop_0.Execute = 0;
				AxisStep = STATE_READY;
			}
			/* check if error occured */
			if (MC_Stop_0.Error == 1)
			{
				GRZAxis.Status.ErrorID = MC_Stop_0.ErrorID;
				MC_Stop_0.Execute = 0;
				AxisStep = STATE_ERROR;
			}
			break;

		/******************** START JOG MOVEMENT POSITVE **********************/
		case STATE_JOG_POSITIVE:  /* STATE: Start jog movement in positive direction */
			MC_MoveVelocity_0.Velocity      = GRZAxis.Parameter.JogVelocity;
			MC_MoveVelocity_0.Acceleration  = GRZAxis.Parameter.Acceleration;
			MC_MoveVelocity_0.Deceleration  = GRZAxis.Parameter.Deceleration;
			MC_MoveVelocity_0.Direction     = mcPOSITIVE_DIR;
			MC_MoveVelocity_0.Execute = 1;
			/* check if jog movement should be stopped */
			if (GRZAxis.Command.MoveJogPos == 0)
			{
				MC_MoveVelocity_0.Execute = 0;
				AxisStep = STATE_HALT;
			}
			/* check if error occured */
			if (MC_MoveVelocity_0.Error == 1)
			{
				GRZAxis.Status.ErrorID = MC_MoveVelocity_0.ErrorID;
				MC_MoveVelocity_0.Execute = 0;
				AxisStep = STATE_ERROR;
			}
			break;

		/******************** START JOG MOVEMENT NEGATIVE **********************/
		case STATE_JOG_NEGATIVE:  /* STATE: Start jog movement in negative direction */
			MC_MoveVelocity_0.Velocity      = GRZAxis.Parameter.JogVelocity;
			MC_MoveVelocity_0.Acceleration  = GRZAxis.Parameter.Acceleration;
			MC_MoveVelocity_0.Deceleration  = GRZAxis.Parameter.Deceleration;
			MC_MoveVelocity_0.Direction     = mcNEGATIVE_DIR;
			MC_MoveVelocity_0.Execute = 1;
			/* check if jog movement should be stopped */
			if (GRZAxis.Command.MoveJogNeg == 0)
			{
				MC_MoveVelocity_0.Execute = 0;
				AxisStep = STATE_HALT;
			}
			/* check if error occured */
			if (MC_MoveVelocity_0.Error == 1)
			{
				GRZAxis.Status.ErrorID = MC_MoveVelocity_0.ErrorID;
				MC_MoveVelocity_0.Execute = 0;
				AxisStep = STATE_ERROR;
			}
			break;

		/******************** START ABSOLUTE MOVEMENT **********************/
		case STATE_MOVE_ABSOLUTE:  /* STATE: Start absolute movement */
			MC_MoveAbsolute_0.Position      = GRZAxis.Parameter.Position;
			MC_MoveAbsolute_0.Velocity      = GRZAxis.Parameter.Velocity;
			MC_MoveAbsolute_0.Acceleration  = GRZAxis.Parameter.Acceleration;
			MC_MoveAbsolute_0.Deceleration  = GRZAxis.Parameter.Deceleration;
			MC_MoveAbsolute_0.Direction     = GRZAxis.Parameter.Direction;
			MC_MoveAbsolute_0.Execute = 1;
			/* check if commanded position is reached */
			if (GRZAxis.Command.Halt == 1)
			{
				GRZAxis.Command.Halt = 0;
				MC_MoveAbsolute_0.Execute = 0;
				AxisStep = STATE_HALT;
			}
			else if (MC_MoveAbsolute_0.Done == 1)
			{
				MC_MoveAbsolute_0.Execute = 0;
				AxisStep = STATE_READY;
			}
			/* check if error occured */
			if (MC_MoveAbsolute_0.Error == 1)
			{
				GRZAxis.Status.ErrorID = MC_MoveAbsolute_0.ErrorID;
				MC_MoveAbsolute_0.Execute = 0;
				AxisStep = STATE_ERROR;
			}
			break;

		/******************** START ADDITIVE MOVEMENT **********************/
		case STATE_MOVE_ADDITIVE:  /* STATE: Start additive movement */
			MC_MoveAdditive_0.Distance      = GRZAxis.Parameter.Distance;
			MC_MoveAdditive_0.Velocity      = GRZAxis.Parameter.Velocity;
			MC_MoveAdditive_0.Acceleration  = GRZAxis.Parameter.Acceleration;
			MC_MoveAdditive_0.Deceleration  = GRZAxis.Parameter.Deceleration;
			MC_MoveAdditive_0.Execute = 1;
			/* check if commanded distance is reached */
			if (GRZAxis.Command.Halt == 1)
			{
				GRZAxis.Command.Halt = 0;
				MC_MoveAdditive_0.Execute = 0;
				AxisStep = STATE_HALT;
			}
			else if (MC_MoveAdditive_0.Done == 1)
			{
				MC_MoveAdditive_0.Execute = 0;
				AxisStep = STATE_READY;
			}
			/* check if error occured */
			if (MC_MoveAdditive_0.Error == 1)
			{
				GRZAxis.Status.ErrorID = MC_MoveAdditive_0.ErrorID;
				MC_MoveAdditive_0.Execute = 0;
				AxisStep = STATE_ERROR;
			}
			break;

		/******************** START VELOCITY MOVEMENT **********************/
		case STATE_MOVE_VELOCITY:  /* STATE: Start velocity movement */
			MC_MoveVelocity_0.Velocity      = GRZAxis.Parameter.Velocity;
			MC_MoveVelocity_0.Acceleration  = GRZAxis.Parameter.Acceleration;
			MC_MoveVelocity_0.Deceleration  = GRZAxis.Parameter.Deceleration;
			MC_MoveVelocity_0.Direction     = GRZAxis.Parameter.Direction;
			MC_MoveVelocity_0.Execute = 1;
			/* check if commanded velocity is reached */
			if (GRZAxis.Command.Halt == 1)
			{
				GRZAxis.Command.Halt = 0;
				MC_MoveVelocity_0.Execute = 0;
				AxisStep = STATE_HALT;
			}
			else if (MC_MoveVelocity_0.InVelocity == 1)
			{
				MC_MoveVelocity_0.Execute = 0;
				AxisStep = STATE_READY;
			}
			/* check if error occured */
			if (MC_MoveVelocity_0.Error == 1)
			{
				GRZAxis.Status.ErrorID = MC_MoveVelocity_0.ErrorID;
				MC_MoveVelocity_0.Execute = 0;
				AxisStep = STATE_ERROR;
			}
			break;

		/******************** FB-ERROR OCCURED *************************/
		case STATE_ERROR:  /* STATE: Error */
			/* check if FB indicates an axis error */
			if (MC_ReadAxisError_0.AxisErrorCount != 0)
			{
				AxisStep = STATE_ERROR_AXIS;
			}
			else
			{
				if (GRZAxis.Command.ErrorAcknowledge == 1)
				{
					GRZAxis.Command.ErrorAcknowledge = 0;
					GRZAxis.Status.ErrorID = 0;
					/* reset axis if it is in axis state ErrorStop */
					if ((MC_ReadStatus_0.Errorstop == 1) && (MC_ReadStatus_0.Valid == 1))
					{
						AxisStep = STATE_ERROR_RESET;
					}
					else
					{
						AxisStep = STATE_WAIT;
					}
				}
			}
			break;

		/******************** AXIS-ERROR OCCURED *************************/
		case STATE_ERROR_AXIS:  /* STATE: Axis Error */
			if (MC_ReadAxisError_0.Valid == 1)
			{
				if (MC_ReadAxisError_0.AxisErrorID != 0)
				{
					GRZAxis.Status.ErrorID = MC_ReadAxisError_0.AxisErrorID;
				}
				MC_ReadAxisError_0.Acknowledge = 0;
				if (GRZAxis.Command.ErrorAcknowledge == 1)
				{
					GRZAxis.Command.ErrorAcknowledge = 0;
					/* acknowledge axis error */
					if (MC_ReadAxisError_0.AxisErrorID != 0)
					{
						MC_ReadAxisError_0.Acknowledge = 1;
					}
				}
				if (MC_ReadAxisError_0.AxisErrorCount == 0)
				{
					GRZAxis.Status.ErrorID = 0;
					/* reset axis if it is in axis state ErrorStop */
					if ((MC_ReadStatus_0.Errorstop == 1) && (MC_ReadStatus_0.Valid == 1))
					{
						AxisStep = STATE_ERROR_RESET;
					}
					else
					{
						AxisStep = STATE_WAIT;
					}
				}
			}
			break;

		/******************** RESET DONE *************************/
		case STATE_ERROR_RESET:  /* STATE: Wait for reset done */
			MC_Reset_0.Execute = 1;
			/* reset MC_Power.Enable if this FB is in Error*/
			if(MC_Power_0.Error == 1)
			{
				MC_Power_0.Enable = 0;
			}
			if(MC_Reset_0.Done == 1)
			{
				MC_Reset_0.Execute = 0;
				AxisStep = STATE_WAIT;
			}
			else if (MC_Reset_0.Error == 1)
			{
				MC_Reset_0.Execute = 0;
				AxisStep = STATE_ERROR;
			}
			break;

		/******************** SEQUENCE END *************************/

		/**********************STATE_READ************************/
		case STATE_READ:
			MC_BR_CyclicRead_0.Enable=1;
			MC_BR_CyclicRead_0.ParID = 277;
			MC_BR_CyclicRead_0.DataAddress = (UDINT)&data;
			MC_BR_CyclicRead_0.DataType =ncPAR_TYP_REAL;

			if (MC_BR_CyclicRead_0.Valid)
			{
				AxisStep = STATE_READY;
			}
			else if (MC_BR_CyclicRead_0.Error)
			{

				GRZAxis.Status.ErrorID = MC_BR_CyclicRead_0.ErrorID;
				/*Reset Enable before going to STATE_ERROR*/
				MC_BR_CyclicRead_0.Enable=0;
				AxisStep = STATE_ERROR;
			}
			break;  /*end read*/

	}

/***************************************************************
        Function Block Calls
***************************************************************/

/************************** MC_POWER ****************************/
	MC_Power_0.Axis = Axis1Obj;  /* pointer to axis */
	MC_Power(&MC_Power_0);

	/************************** MC_HOME *****************************/
	MC_Home_0.Axis = Axis1Obj;
	MC_Home(&MC_Home_0);

	/********************** MC_MOVEABSOLUTE *************************/
	MC_MoveAbsolute_0.Axis = Axis1Obj;
	MC_MoveAbsolute(&MC_MoveAbsolute_0);

	/********************** MC_MOVEADDITIVE *************************/
	MC_MoveAdditive_0.Axis = Axis1Obj;
	MC_MoveAdditive(&MC_MoveAdditive_0);

	/********************** MC_MOVEVELOCITY *************************/
	MC_MoveVelocity_0.Axis = Axis1Obj;
	MC_MoveVelocity(&MC_MoveVelocity_0);

	/************************** MC_STOP *****************************/
	MC_Stop_0.Axis = Axis1Obj;
	MC_Stop(&MC_Stop_0);

	/**************************MC_HALT*******************************/
	MC_Halt_0.Axis = Axis1Obj;
	MC_Halt(&MC_Halt_0);

	/************************** MC_RESET ****************************/
	MC_Reset_0.Axis = Axis1Obj;
	MC_Reset(&MC_Reset_0);

	MC_BR_CyclicRead_0.Axis = Axis1Obj;
	MC_BR_CyclicRead(&MC_BR_CyclicRead_0);

}
```

- LazerMarkalama.opct - A new OPC tag file. (not shown)

### Package Logical/LibDVFrame1_ST - Read and write serial Frames

### Program Logical/LibDVFrame1_ST/Sender (IEC) - sending serial data

#### SenderCyclic.st - Cyclic code
```iecst
(********************************************************************
 * COPYRIGHT -- Bernecker + Rainer
 ********************************************************************
 * Program: Sender
 * File: SenderCyclic.st
 * Author: Bernecker & Rainer
 * Created: January 25, 2010
 ********************************************************************
 * Implementation of program Sender
 ********************************************************************)

(*************init program**********************)
PROGRAM _INIT
	Sender.Commands.open_send := FALSE;												(*enable sender by default*)
END_PROGRAM

(*************cyclic program********************)
PROGRAM _CYCLIC

	CASE Sender.step OF
		FRM_WAIT:	(*--- wait for command*)

			IF Sender.Commands.open_send = TRUE THEN								(*command for sender activation*)
				Sender.step := FRM_OPEN;
   			END_IF

			(*close will be requested in step FRM_WRITE*)

		FRM_OPEN:	(*--- open serial interface*)

			(*Parameters for FRM_xopen()*)
			Sender.FRM_xopen_0.enable := TRUE;
			Sender.FRM_xopen_0.device := ADR('IF1');										(*Devicename --> see your serial interface properties*)
			Sender.FRM_xopen_0.mode := ADR('/PHY=RS232 /BD=9600 /DB=8 /PA=N /SB=1'); 		(*Modestring --> specifies the seria operation mode*)
			Sender.FRM_xopen_0.config := ADR(Sender.xopenConfig) ;					(*Additional Parameters, optional*)

			(*Additional Parameters for FRM_xopen()*)
			Sender.xopenConfig.idle := 10;											(*Idle time between two characters*)
			Sender.xopenConfig.delimc := 0;											(*activate two delimeters*)
			Sender.xopenConfig.delim[0] := 0; 										(*CR - carridge return -> dec 13*)
			Sender.xopenConfig.delim[1] := 0; 										(*LF - line feed -> dec 10*)
			Sender.xopenConfig.tx_cnt := 3;											(*number of transmit buffers*)
			Sender.xopenConfig.rx_cnt := 3; 										(*number of receive buffers*)
			Sender.xopenConfig.tx_len := 256; 										(*length of transmit buffers*)
			Sender.xopenConfig.rx_len := 256; 										(*lenght of receive buffers*)
			Sender.xopenConfig.argc := 0;											(*activate additional options*)
			Sender.xopenConfig.argv := 0;											(*parameters for additional options (check help)*)

			Sender.FRM_xopen_0();													(*call the FRM_xopen() function*)

			IF Sender.FRM_xopen_0.status = 0 THEN
				Sender.step := FRM_GBUF;											(*Interface opend successfully --> next step*)
			ELSIF Sender.FRM_xopen_0.status = BUSY THEN
				Sender.step := FRM_OPEN;											(*operation not finished yet --> call again*)
			ELSE
				Sender.step := FRM_ERROR;											(*function returned errorcode --> check help*)
   			END_IF

		FRM_GBUF:	(*--- aquire sendbuffer for FRM_WRITE*)
			Sender.FRM_gbuf_0.enable := TRUE;
   			Sender.FRM_gbuf_0.ident := Sender.FRM_xopen_0.ident;

			Sender.FRM_gbuf_0();													(*call the FRM_gbuf() function*)

			IF Sender.FRM_gbuf_0.status = 0 THEN
				memset(Sender.FRM_gbuf_0.buffer,0,Sender.FRM_gbuf_0.buflng);		(*clear sendbuffer*)
				Sender.step := FRM_PREPARE_SENDDATA;								(*system returned a valid buffer --> next step*)
			ELSIF Sender.FRM_gbuf_0.status = BUSY THEN
				Sender.step := FRM_GBUF;											(*operation not finished yet --> call again*)
			ELSE
				Sender.step := FRM_ERROR;											(*function returned errorcode --> check help*)
   			END_IF

		FRM_PREPARE_SENDDATA: (*--- prepare senddata, copy data to sendbuffer*)

			counterUp := counterUp + 1;												(*simulate counter up*)

			itoa(UINT_TO_DINT(counterUp),ADR(helpString));							(*convert data to string*)

			Sender.send_data := 'INIT';
			strcat(ADR(Sender.send_data),ADR(helpString));							(*attach value*)
			strcat(ADR(Sender.send_data),ADR('$R$L'));								(*attach CR + LF*)

			strcpy(Sender.FRM_gbuf_0.buffer,ADR(Sender.send_data));					(*copy senddata to sendbuffer*)

			Sender.step := FRM_WRITE;												(*--> next step*)

		FRM_WRITE:	(*--- write data to interface*)

			(*Parameters for FRM_write()*)
			Sender.FRM_write_0.enable := TRUE;
			Sender.FRM_write_0.ident := Sender.FRM_xopen_0.ident;					(*ident from FRM_xopen()*)
			Sender.FRM_write_0.buffer := Sender.FRM_gbuf_0.buffer;					(*sendbuffer*)
			Sender.FRM_write_0.buflng := strlen(ADR(Sender.send_data));				(*net length of senddata*)

			Sender.FRM_write_0();													(*call the FRM_write() function*)

			IF Sender.FRM_write_0.status = 0 THEN
				IF Sender.Commands.close = TRUE THEN								(*requst to close the serial port*)
					Sender.Commands.open_send := FALSE;								(*disable command open_send*)
					Sender.step := FRM_CLOSE;
				ELSE
					Sender.step := FRM_GBUF;										(*writing successful --> get next sendbuffer*)
				END_IF
			ELSIF Sender.FRM_write_0.status = BUSY THEN
				Sender.step := FRM_WRITE;											(*operation not finished yet --> call again*)
			ELSE
				Sender.step := FRM_ROBUF;											(*function returned errorcode --> check help*)
   			END_IF

		FRM_ROBUF:	(*--- release sendbuffer in case of no successful write operation*)
			Sender.FRM_robuf_0.enable := TRUE;
			Sender.FRM_robuf_0.buffer := Sender.FRM_gbuf_0.buffer;					(*sendbuffer*)
			Sender.FRM_robuf_0.buflng := Sender.FRM_gbuf_0.buflng;					(*buffer length*)

			Sender.FRM_robuf_0();													(*call the FRM_robuf() function*)

			IF Sender.FRM_robuf_0.status = 0 THEN
				Sender.step := FRM_GBUF;											(*released buffer successful --> get next sendbuffer*)
			ELSIF Sender.FRM_robuf_0.status = BUSY THEN
				Sender.step := FRM_ROBUF;											(*operation not finished yet --> call again*)
			ELSE
				Sender.step := FRM_ERROR;											(*function returned errorcode --> check help*)
   			END_IF

		FRM_CLOSE:	(*--- close the interface*)
			Sender.FRM_close_0.enable := TRUE;
   			Sender.FRM_close_0.ident := Sender.FRM_xopen_0.ident;					(*ident from FRM_xopen()*)

			Sender.FRM_close_0();													(*call the FRM_close() function*)

			IF Sender.FRM_close_0.status = 0 THEN
				Sender.Commands.close := FALSE;										(*disable close command*)
				Sender.step := FRM_WAIT;											(*closed interface successfully --> wait step*)
			ELSIF Sender.FRM_close_0.status = BUSY THEN
				Sender.step := FRM_CLOSE;											(*operation not finished yet --> call again*)
			ELSE
				Sender.step := FRM_ERROR;											(*function returned errorcode --> check help*)
			END_IF

		FRM_ERROR:	(*--- error handling*)
			; (*not implementet yet, check help for error codes*)
 	END_CASE

END_PROGRAM
```

#### Sender.typ - Local data types
```iecst
(********************************************************************
 * COPYRIGHT -- Bernecker + Rainer
 ********************************************************************
 * Program: Sender
 * File: Sender.typ
 * Author: Bernecker & Rainer
 * Created: January 25, 2010
 ********************************************************************
 * Local data types of program Sender
 ********************************************************************)
(*Enumeration for Statemachine*)

TYPE
	enSEND_STEPS :
		(
		FRM_WAIT := 0, (*Defines the wait step*)
		FRM_OPEN, (*Defines Step for FRM_xopen() *)
		FRM_GBUF, (*Defines Step for FRM_rbuf()*)
		FRM_PREPARE_SENDDATA, (*Defines Step for preparing send data*)
		FRM_WRITE, (*Defines Step for FRM_write()*)
		FRM_ROBUF, (*Defines Step for FRM_robuf()*)
		FRM_CLOSE, (*Defines Step for FRM_close()*)
		FRM_ERROR := 255 (*Defines Step for Errorhandling*)
		);
END_TYPE

(*Command data type*)

TYPE
	command_typ : 	STRUCT
		open_send : BOOL; (*Open serial port and send data*)
		close : BOOL; (*Close serial port*)
	END_STRUCT;
END_TYPE

(*Sender type*)

TYPE
	Sender_typ : 	STRUCT
		step : enSEND_STEPS := FRM_OPEN; (*Step of the Statemachine*)
		Commands : command_typ; (*Commandinterface*)
		send_data : STRING[80]; (*Send data*)
		FRM_xopen_0 : FRM_xopen; (*Functionblock FRM_xopen()*)
		xopenConfig : XOPENCONFIG; (*Configuration Type for FRM_xopen()*)
		FRM_gbuf_0 : FRM_gbuf; (*Functionblock FRM_gbuf()*)
		FRM_robuf_0 : FRM_robuf; (*Functionblock FRM_robuf()*)
		FRM_write_0 : FRM_write; (*Functionblock FRM_write)*)
		FRM_close_0 : FRM_close; (*Functionblock FRM_close()*)
	END_STRUCT;
END_TYPE
```

#### Sender.var - Local variables
```iecst
(********************************************************************
 * COPYRIGHT -- Bernecker + Rainer
 ********************************************************************
 * Program: Sender
 * File: Sender.var
 * Author: Bernecker & Rainer
 * Created: January 25, 2010
 ********************************************************************
 * Local variables of program Sender
 ********************************************************************)
VAR
	Sender : Sender_typ := (0); (*Structure with all instances and variables*)
END_VAR
VAR CONSTANT
	BUSY : UINT := 65535; (*Functionblock BUSY status*)
END_VAR
VAR
	counterUp : UINT; (*Simulation of counter up*)
	helpString : STRING[80]; (*helpstring for integer to ascii conversion*)
END_VAR
```

### Program Logical/LibDVFrame1_ST/Receiver (IEC) - receiving serial data

#### ReceiverCyclic.st - Cyclic code
```iecst
(********************************************************************
 * COPYRIGHT -- Bernecker + Rainer
 ********************************************************************
 * Program: Receiver
 * File: ReceiverCyclic.st
 * Author: Bernecker & Rainer
 * Created: January 25, 2010
 ********************************************************************
 * Implementation of program Receiver
 ********************************************************************)

(*************init program**********************)
PROGRAM _INIT
	Receiver.Commands.open_receive := TRUE;												(*enable Receiver by default*)
END_PROGRAM

(*************cyclic program********************)
PROGRAM _CYCLIC

	CASE Receiver.step OF
		FRM_WAIT:	(*--- wait for command*)

			IF Receiver.Commands.open_receive = TRUE THEN								(*command for Receiver activation*)
				Receiver.step := FRM_OPEN;
   			END_IF

			(*close will be requested in step FRM_RBUF*)

		FRM_OPEN:	(*--- open serial interface*)

			(*Parameters for FRM_xopen()*)
			Receiver.FRM_xopen_0.enable := TRUE;
			Receiver.FRM_xopen_0.device := ADR('IF1');							(*Devicename --> see your serial interface properties*)
			Receiver.FRM_xopen_0.mode := ADR('/PHY=RS232 /BD=9600 /DB=8 /PA=N /SB=1'); (*Modestring --> specifies the seria operation mode*)
			Receiver.FRM_xopen_0.config := ADR(Receiver.xopenConfig) ;					(*Additional Parameters, optional*)

			(*Additional Parameters for FRM_xopen()*)
			Receiver.xopenConfig.idle := 10;											(*Idle time between two characters*)
			Receiver.xopenConfig.delimc := 0;											(*activate two delimeters*)
			Receiver.xopenConfig.delim[0] := 0; 										(*e.g. CR - carridge return -> dec 13*)
			Receiver.xopenConfig.delim[1] := 0; 										(*e.g. LF - line feed -> dec 10*)
			Receiver.xopenConfig.tx_cnt := 3;											(*number of transmit buffers*)
			Receiver.xopenConfig.rx_cnt := 3; 											(*number of receive buffers*)
			Receiver.xopenConfig.tx_len := 256; 										(*length of transmit buffers*)
			Receiver.xopenConfig.rx_len := 256; 										(*lenght of receive buffers*)
			Receiver.xopenConfig.argc := 0;												(*activate additional options*)
			Receiver.xopenConfig.argv := 0;												(*parameters for additional options (check help)*)

			Receiver.FRM_xopen_0();														(*call the FRM_xopen() function*)

			IF Receiver.FRM_xopen_0.status = 0 THEN
				Receiver.step := FRM_READ;												(*Interface opend successfully --> next step*)
			ELSIF Receiver.FRM_xopen_0.status = BUSY THEN
				Receiver.step := FRM_OPEN;												(*operation not finished yet --> call again*)
			ELSE
				Receiver.step := FRM_ERROR;												(*function returned errorcode --> check help*)
   			END_IF

		FRM_READ:	(*--- read data from serial interface*)
			Receiver.FRM_read_0.enable := TRUE;
   			Receiver.FRM_read_0.ident := Receiver.FRM_xopen_0.ident;

			Receiver.FRM_read_0();														(*call the FRM_read() function*)

			IF Receiver.FRM_read_0.status = 0 THEN
				Receiver.step := FRM_COPY_RD_DATA;										(*system returned a valid data --> next step*)
			ELSIF Receiver.FRM_read_0.status = frmERR_NOINPUT THEN
				Receiver.step := FRM_READ;												(*no data available --> call again*)
			ELSIF Receiver.FRM_read_0.status = frmERR_INPUTERROR THEN
				Receiver.step := FRM_RBUF;												(*received Frame with defective characters, skip data*)
			ELSE
				Receiver.step := FRM_ERROR;												(*function returned errorcode --> check help*)
   			END_IF

		FRM_COPY_RD_DATA: (*--- copy data out of the receive buffer*)
			memset(ADR(Receiver.receive_data),0,SIZEOF(Receiver.receive_data));			(*clear read_data buffer*)
			memcpy(ADR(Receiver.receive_data),Receiver.FRM_read_0.buffer,Receiver.FRM_read_0.buflng);     (*copy and evaluate read data*)
			Receiver.step := FRM_RBUF;													(*release read buffer*)

		FRM_RBUF:	(*--- release readbuffer*)

			(*Parameters for FRM_rbuf()*)
			Receiver.FRM_rbuf_0.enable := TRUE;
			Receiver.FRM_rbuf_0.ident := Receiver.FRM_xopen_0.ident;					(*ident from FRM_xopen()*)
			Receiver.FRM_rbuf_0.buffer := Receiver.FRM_read_0.buffer;					(*read buffer*)
			Receiver.FRM_rbuf_0.buflng := Receiver.FRM_read_0.buflng;					(*length of sendbuffer*)

			Receiver.FRM_rbuf_0();														(*call the FRM_rbuf() function*)

			IF Receiver.FRM_rbuf_0.status = 0 THEN
				IF Receiver.Commands.close = TRUE THEN
					Receiver.Commands.open_receive := FALSE;								(*disable command open_send*)
					Receiver.step := FRM_CLOSE;											(*request to close serial port*)
				ELSE
					Receiver.step := FRM_READ;											(*read again*)
				END_IF
			ELSIF Receiver.FRM_rbuf_0.status = BUSY THEN
				Receiver.step := FRM_RBUF;												(*operation not finished yet --> call again*)
			ELSIF Receiver.FRM_rbuf_0.status = frmERR_INVALIDBUFFER THEN
				Receiver.step := FRM_READ;												(*buffer is invalid --> read again*)
			ELSE
				Receiver.step := FRM_ERROR;												(*function returned errorcode --> check help*)
   			END_IF

		FRM_CLOSE:	(*--- close the interface*)
			Receiver.FRM_close_0.enable := TRUE;
   			Receiver.FRM_close_0.ident := Receiver.FRM_xopen_0.ident;					(*ident from FRM_xopen()*)

			Receiver.FRM_close_0();														(*call the FRM_close() function*)

			IF Receiver.FRM_close_0.status = 0 THEN
				Receiver.Commands.close := FALSE;										(*disable close command*)
				Receiver.step := FRM_WAIT;												(*closed interface successfully --> wait step*)
			ELSIF Receiver.FRM_close_0.status = BUSY THEN
				Receiver.step := FRM_CLOSE;												(*operation not finished yet --> call again*)
			ELSE
				Receiver.step := FRM_ERROR;												(*function returned errorcode --> check help*)
			END_IF

		FRM_ERROR:	(*--- error handling*)
			; (*not implementet yet, check help for error codes*)
 	END_CASE

END_PROGRAM
```

#### Receiver.typ - Local data types
```iecst
(********************************************************************
 * COPYRIGHT -- Bernecker + Rainer
 ********************************************************************
 * Program: Receiver
 * File: Receiver.typ
 * Author: Bernecker & Rainer
 * Created: January 25, 2010
 ********************************************************************
 * Local data types of program Receiver
 ********************************************************************)
(*Enumeration for Statemachine*)

TYPE
	enRECV_STEPS :
		(
		FRM_WAIT := 0, (*Defines the wait step*)
		FRM_OPEN, (*Defines Step for FRM_xopen() *)
		FRM_READ, (*Defines Step for FRM_read()*)
		FRM_COPY_RD_DATA, (*Defines Step for storing read data*)
		FRM_RBUF, (*Defines Step for FRM_rbuf()*)
		FRM_CLOSE, (*Defines Step for FRM_close()*)
		FRM_ERROR := 255 (*Defines Step for Errorhandling*)
		);
END_TYPE

(*Command data type*)

TYPE
	command_typ : 	STRUCT
		open_receive : BOOL; (*Open serial port and receive data*)
		close : BOOL; (*Close serial port*)
	END_STRUCT;
END_TYPE

(*Receiver type*)

TYPE
	Receiver_typ : 	STRUCT
		step : enRECV_STEPS; (*Step of the Statemachine*)
		Commands : command_typ; (*Commandinterface*)
		receive_data : STRING[80]; (*receive data*)
		FRM_xopen_0 : FRM_xopen; (*Functionblock FRM_xopen()*)
		xopenConfig : XOPENCONFIG; (*Configuration Type for FRM_xopen()*)
		FRM_read_0 : FRM_read; (*Functionblock FRM_read()*)
		FRM_rbuf_0 : FRM_rbuf; (*Functionblock FRM_rbuf()*)
		FRM_close_0 : FRM_close; (*Functionblock FRM_close()*)
	END_STRUCT;
END_TYPE
```

#### Receiver.var - Local variables
```iecst
(********************************************************************
 * COPYRIGHT -- Bernecker + Rainer
 ********************************************************************
 * Program: Sender
 * File: Sender.var
 * Author: Bernecker & Rainer
 * Created: January 25, 2010
 ********************************************************************
 * Local variables of program Sender
 ********************************************************************)
VAR
	Receiver : Receiver_typ := (0); (*local Struktur with all instances and variables*)
END_VAR
VAR CONSTANT
	BUSY : UINT := 65535; (*Functionblock BUSY status*)
END_VAR
```

Listed in the project but not available here: Logical/RZAxisobj/gz1_axisa, Logical/RC1Axisobj/gc2_axisa, Logical/RC2Axisobj/gc2_axisa, Logical/Master/edge.h, Logical/PowerAx1/PowerAx1.typ, Logical/PowerAx1/PowerAx1.var, Logical/PowerAx1/edge.h, Logical/PowerAx2/PowerAx2.typ, Logical/PowerAx2/PowerAx2.var, Logical/PowerAx2/edge.h, Logical/RAAxisControl/GX1Ax.typ, Logical/RAAxisControl/edge.h, Logical/RXAxisControl/GX2Ax.typ, Logical/RXAxisControl/GX2Ax.var, Logical/RXAxisControl/edge.h, Logical/RYAxisControl/GX3Ax.typ, Logical/RYAxisControl/GX3Ax.var, Logical/RYAxisControl/edge.h, Logical/RZAxisControl/GZ1Ax.typ, Logical/RZAxisControl/edge.h, Logical/RC1AxisControl/GC1Ax.typ, Logical/RC1AxisControl/GC1Ax.var, Logical/RC1AxisControl/edge.h, Logical/RC2AxisControl/GC2Ax.typ, Logical/RC2AxisControl/edge.h, Logical/GRXAxisControl/GRXAx.typ, Logical/GRXAxisControl/GRXAx.var, Logical/GRXAxisControl/edge.h, Logical/GRZAxisControl/GRXAx.var, Logical/GRZAxisControl/edge.h
